// Mitsubishi GX Works2 project: 0129 실린더1개 편솔 레더   PLC: Q03UDV

PROGRAM MAIN
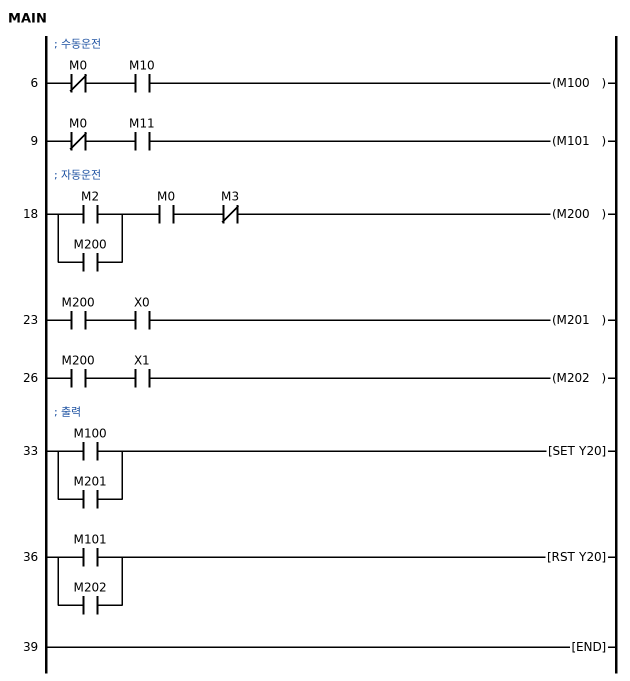
; 수동운전
6     LDI     M0
      AND     M10
      OUT     M100
9     LDI     M0
      AND     M11
      OUT     M101
; 자동운전
18    LD      M2
      OR      M200
      AND     M0
      ANI     M3
      OUT     M200
23    LD      M200
      AND     X0
      OUT     M201
26    LD      M200
      AND     X1
      OUT     M202
; 출력
33    LD      M100
      OR      M201
      SET     Y20
36    LD      M101
      OR      M202
      RST     Y20
39    END
END_PROGRAM
